{region '#Template'}
	{attribute 'Category' := 'Universal'}
	{attribute 'Version' := '0.0.1.0'}
	{attribute 'Tags' := 'Universal, Valve'}
	{attribute 'Description' := 'Ventil analog	// Valve analog'}
{endregion}
FUNCTION_BLOCK FB_BA_Vlv EXTENDS FB_BA_ActuatorAnalog
VAR_INPUT
	bAblkLock				: BOOL;
END_VAR
VAR_OUTPUT
END_VAR
VAR_INPUT CONSTANT
	Ablk					: FB_BA_AntiBlocking;	
	Fdb						: FB_BA_AI_IO;		 
END_VAR

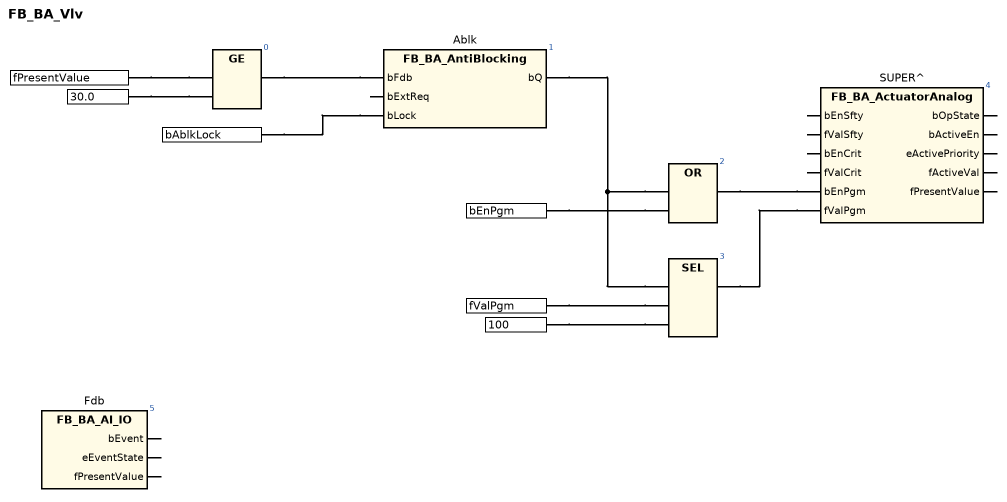
Ablk(bFdb := fPresentValue >= 30.0, bLock := bAblkLock); // FB_BA_AntiBlocking
SUPER^(bEnPgm := Ablk.bQ OR bEnPgm, fValPgm := SEL(Ablk.bQ, fValPgm, 100)); // FB_BA_ActuatorAnalog
Fdb(); // FB_BA_AI_IO

METHOD FB_init : BOOL
VAR_INPUT
	bInitRetains : BOOL; // if TRUE, the retain variables are initialized (warm start / cold start)
	bInCopyCode : BOOL;  // if TRUE, the instance afterwards gets moved into the copy code (online change)
END_VAR
Ablk.iParent					:= THIS^;	
Ablk.iLabel						:= LblUniFieldDevice.Valve_Ablk;
Ablk.sObjectName				:= '{Idx=01}';																	
Ablk.eDPADMode					:= E_BA_DPADMode.eIncludeDescription;	

Fdb.iParent						:= THIS^;		
Fdb.iLabel 						:= LblUniFieldDevice.Valve_Fdb;
Fdb.sObjectName					:= '{Idx=01}';
Fdb.sDeviceType					:= '';
Fdb.bEnOutOfService				:= FALSE;
Fdb.eUnit						:= E_BA_Unit.eOther_Percent;
Fdb.fResolution 				:= 0.03051851;
Fdb.fScaleOffset 				:= 0; 	
Fdb.fCOVIncrement				:= BA2_Param.fDefCOVIncrement;
Fdb.nEventClassID				:= EventClasses.OtherSimple;
Fdb.stTimeDelay.nToNormal		:= BA2_Param.nDefTimeDelay_ToNormal;
Fdb.stTimeDelay.nToAbnormal		:= BA2_Param.nDefTimeDelay_ToAbnormal;
Fdb.stHighLimit.bEnable			:= FALSE;
Fdb.stHighLimit.fValue			:= 0.0;		
Fdb.stLowLimit.bEnable			:= FALSE;
Fdb.stLowLimit.fValue			:= 0.0;
Fdb.fLimitDeadband 				:= BA2_Param.fDefLimitDeadband;
Fdb.bAcknowledgeRm				:= FALSE;	
Fdb.aEventTransitionText[1]		:= Texts.txtExceeded;
Fdb.aEventTransitionText[2]		:= Texts.txtDisturb;
Fdb.aEventTransitionText[3]		:= Texts.txtNormal;
Fdb.bEventDetectionEnable		:= FALSE;
Fdb.eEnPlantLock				:= E_BA_LockPriority.eNoLock;
END_METHOD

END_FUNCTION_BLOCK

(* stored: Version 1.1.0.1, ProductVersion 3.1.4024.6
   POU FB_BA_Vlv: Id {dacde8ae-c826-474b-9152-26b72cbd594c}, SpecialFunc None
   Method FB_init: Id {a2ce6982-f36d-48e0-92fd-30eb731612f6} *)
